{attribute 'qualified_only'}
VAR_GLOBAL
	// COMMUNICATION variables
	ReceivedStringArray : ARRAY[0..200] OF STRING;
	ReceivedStringWordCounter : INT := 0;

	ReceivedCMD : STRING := '';
	VarValue : STRING := '';
	VarType : STRING := '';
	VarName : STRING := '';
	//
END_VAR

(* stored: Version 1.1.0.1, ProductVersion 3.1.4024.12
   GVL GVL: Id {a4a1f3b6-3430-4b84-b16b-3f00b70af1b1} *)
